{attribute 'qualified_only'}
{attribute 'strict'}
TYPE E_ButtonSelection :
(
	Tap := 0,		//	toggle if Event rising edge is detected
	Toggle := 1		//	0: off | 1: on
);
END_TYPE

(* stored: Version 1.1.0.1, ProductVersion 3.1.4024.12
   DUT E_ButtonSelection: Id {eae2fb99-bc36-498d-afa8-9a6bc50b6b63} *)
